(* CODESYS project Uppgift 9 - lösning 2.project

Project tree, tasks and I/O mapping:
  Device : CODESYS Control Win V3, 3S - Smart Software Solutions GmbH, order no. 305021, version 3.5.10.40
    application Application
      libraries: Standard, * (System)
      task MainTask (cyclic, interval t#20ms, priority 1) calls PLC_PRG
      program PLC_PRG [LD]
*)

// Device/Application/PLC_PRG
PROGRAM PLC_PRG
VAR
	TON_0: TON;
	TON_1: TON;
	Yellow_Lamp: BOOL;
	Btn_1: BOOL;
	Blue_lamp: BOOL;
	Green_Lamp: BOOL;
	TON_2: TON;
	Output_1: TIME;
	Output_2: TIME;
	Output_3: TIME;
END_VAR

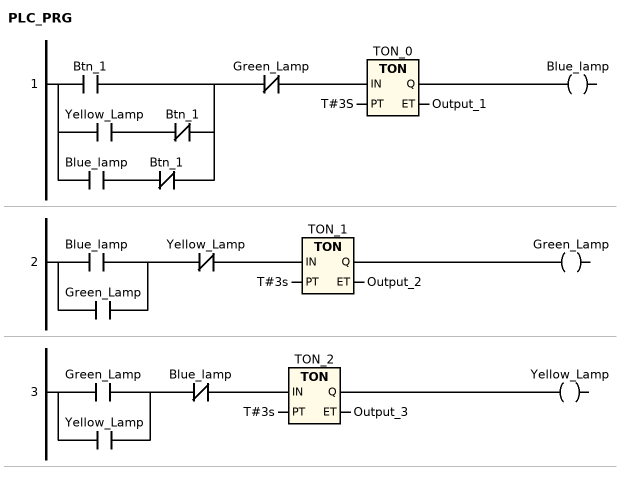
// NETWORK 1
TON_0(
    IN := (Btn_1 OR Yellow_Lamp AND NOT Btn_1 OR Blue_lamp AND NOT Btn_1) AND NOT Green_Lamp,
    PT := T#3S,
    ET => Output_1); // TON
Blue_lamp := TON_0.Q;

// NETWORK 2
TON_1(IN := (Blue_lamp OR Green_Lamp) AND NOT Yellow_Lamp, PT := T#3s, ET => Output_2); // TON
Green_Lamp := TON_1.Q;

// NETWORK 3
TON_2(IN := (Green_Lamp OR Yellow_Lamp) AND NOT Blue_lamp, PT := T#3s, ET => Output_3); // TON
Yellow_Lamp := TON_2.Q;

END_PROGRAM
